TYPE T_InstancePath : STRING(512); END_TYPE

(* stored: Version 1.1.0.1, ProductVersion 3.1.4024.12
   DUT T_InstancePath: Id {27ede6f0-26cf-46a3-8a99-767f929d8da6} *)
